FUNCTION_BLOCK SBSensorRC (* Sensor for a Sonnenbatterie via its RESTful API. *)
  (* Standard: 61499-2; Description: Requires the http communication layer. This function block makes use of CLNTRC FBs (see Utils subdirectory of this library) instead of CLIENT FBs. *)
  (* Version 1.0, 2017-08-27, Marc Jakobi, HTW Berlin *)
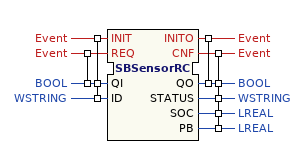
  EVENT_INPUT
    INIT WITH QI, ID; (* Initialization Request *)
    REQ WITH QI; (* Normal Execution Request *)
  END_EVENT
  EVENT_OUTPUT
    INITO WITH QO; (* Initialization Confirm *)
    CNF WITH QO, STATUS, SOC, PB; (* Execution Confirmation *)
  END_EVENT
  VAR_INPUT
    QI : BOOL; (* Input event qualifier *)
    ID : WSTRING; (* Connection identifier (ip:port) *)
  END_VAR
  VAR_OUTPUT
    QO : BOOL; (* Output event qualifier *)
    STATUS : WSTRING; (* HTTP response codes *)
    SOC : LREAL; (* State of charge [0,..,1] *)
    PB : LREAL; (* Battery transfer (positive = charge, negative = discharge) in W *)
  END_VAR
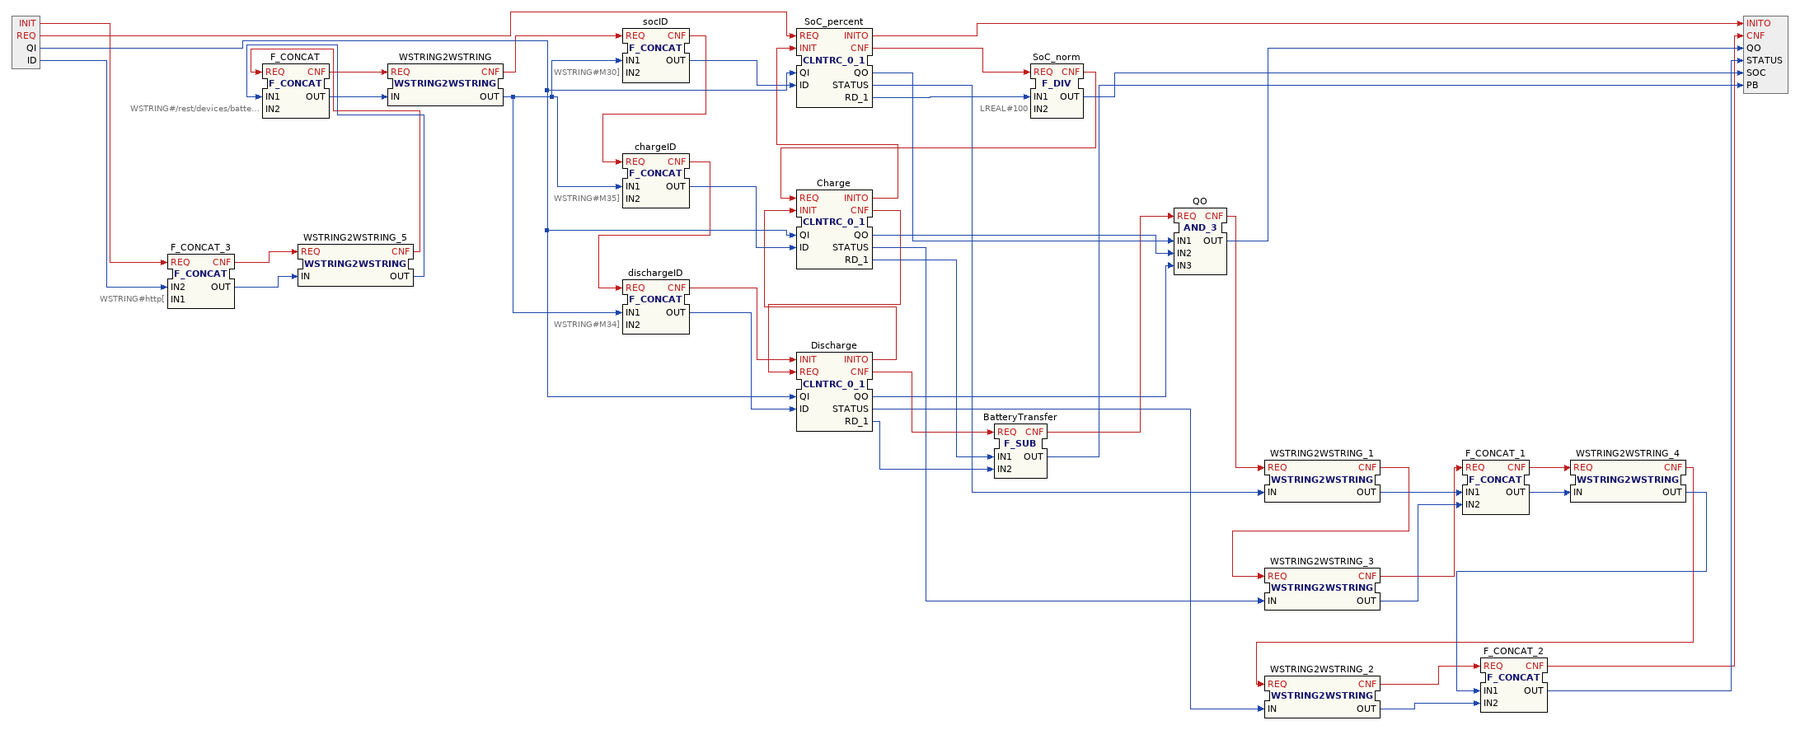
  FBS
    WSTRING2WSTRING : WSTRING2WSTRING;
    F_CONCAT : F_CONCAT(IN2 := WSTRING#/rest/devices/battery/);
    socID : F_CONCAT(IN2 := WSTRING#M30]);
    chargeID : F_CONCAT(IN2 := WSTRING#M35]);
    dischargeID : F_CONCAT(IN2 := WSTRING#M34]);
    QO : AND_3;
    SoC_norm : F_DIV(IN2 := LREAL#100);
    BatteryTransfer : F_SUB;
    WSTRING2WSTRING_1 : WSTRING2WSTRING;
    WSTRING2WSTRING_2 : WSTRING2WSTRING;
    WSTRING2WSTRING_3 : WSTRING2WSTRING;
    WSTRING2WSTRING_4 : WSTRING2WSTRING;
    F_CONCAT_1 : F_CONCAT;
    F_CONCAT_2 : F_CONCAT;
    F_CONCAT_3 : F_CONCAT(IN1 := WSTRING#http[);
    WSTRING2WSTRING_5 : WSTRING2WSTRING;
    SoC_percent : CLNTRC_0_1;
    Charge : CLNTRC_0_1;
    Discharge : CLNTRC_0_1;
  END_FBS
  EVENT_CONNECTIONS
    WSTRING2WSTRING.CNF TO socID.REQ;
    socID.CNF TO chargeID.REQ;
    chargeID.CNF TO dischargeID.REQ;
    QO.CNF TO WSTRING2WSTRING_1.REQ;
    WSTRING2WSTRING_1.CNF TO WSTRING2WSTRING_3.REQ;
    WSTRING2WSTRING_3.CNF TO F_CONCAT_1.REQ;
    F_CONCAT_1.CNF TO WSTRING2WSTRING_4.REQ;
    WSTRING2WSTRING_4.CNF TO WSTRING2WSTRING_2.REQ;
    WSTRING2WSTRING_2.CNF TO F_CONCAT_2.REQ;
    F_CONCAT_2.CNF TO CNF;
    INIT TO F_CONCAT_3.REQ;
    F_CONCAT.CNF TO WSTRING2WSTRING.REQ;
    F_CONCAT_3.CNF TO WSTRING2WSTRING_5.REQ;
    WSTRING2WSTRING_5.CNF TO F_CONCAT.REQ;
    BatteryTransfer.CNF TO QO.REQ;
    REQ TO SoC_percent.REQ;
    SoC_percent.INITO TO INITO;
    SoC_percent.CNF TO SoC_norm.REQ;
    SoC_norm.CNF TO Charge.REQ;
    Charge.INITO TO SoC_percent.INIT;
    dischargeID.CNF TO Discharge.INIT;
    Charge.CNF TO Discharge.REQ;
    Discharge.INITO TO Charge.INIT;
    Discharge.CNF TO BatteryTransfer.REQ;
  END_CONNECTIONS
  DATA_CONNECTIONS
    WSTRING2WSTRING.OUT TO socID.IN1;
    WSTRING2WSTRING.OUT TO chargeID.IN1;
    SoC_norm.OUT TO SOC;
    BatteryTransfer.OUT TO PB;
    QO.OUT TO QO;
    WSTRING2WSTRING_1.OUT TO F_CONCAT_1.IN1;
    WSTRING2WSTRING_3.OUT TO F_CONCAT_1.IN2;
    F_CONCAT_1.OUT TO WSTRING2WSTRING_4.IN;
    WSTRING2WSTRING_4.OUT TO F_CONCAT_2.IN1;
    WSTRING2WSTRING_2.OUT TO F_CONCAT_2.IN2;
    F_CONCAT_2.OUT TO STATUS;
    WSTRING2WSTRING.OUT TO dischargeID.IN1;
    ID TO F_CONCAT_3.IN2;
    F_CONCAT.OUT TO WSTRING2WSTRING.IN;
    F_CONCAT_3.OUT TO WSTRING2WSTRING_5.IN;
    WSTRING2WSTRING_5.OUT TO F_CONCAT.IN1;
    QI TO SoC_percent.QI;
    socID.OUT TO SoC_percent.ID;
    SoC_percent.QO TO QO.IN1;
    SoC_percent.STATUS TO WSTRING2WSTRING_1.IN;
    SoC_percent.RD_1 TO SoC_norm.IN1;
    QI TO Charge.QI;
    chargeID.OUT TO Charge.ID;
    Charge.QO TO QO.IN2;
    Charge.STATUS TO WSTRING2WSTRING_3.IN;
    Charge.RD_1 TO BatteryTransfer.IN1;
    QI TO Discharge.QI;
    dischargeID.OUT TO Discharge.ID;
    Discharge.QO TO QO.IN3;
    Discharge.STATUS TO WSTRING2WSTRING_2.IN;
    Discharge.RD_1 TO BatteryTransfer.IN2;
  END_CONNECTIONS
END_FUNCTION_BLOCK
